{attribute addProperty BoxType "EL3314-0030-0021"}
{attribute addProperty Id "StatusAT %I*Status_C3A5DD7C1621ValueAT %I*DINT32417"}
{attribute addProperty CRC "1202977787"}
{attribute addProperty SizeInBites "48"}
{attribute addProperty SizeInBytes "6"}
TYPE TC_Inputs_Channel_47B3FBFB :
STRUCT
	{attribute addProperty Name "Status"}
	Status AT %I* : Status_C3A5DD7C;
	{attribute addProperty Name "Value"}
	Value AT %I* : DINT;
END_STRUCT
END_TYPE

(* stored: Version 1.2.0.0, ProductVersion 3.1.4024.9
   DUT TC_Inputs_Channel_47B3FBFB: Id {155de5c0-5def-4008-85cb-98016f453dd2} *)
